PROGRAM prg_Verschalingmetfunctie
VAR
	//POTENTIOMETERRRR
	//0 tot 32767
	nPotentiometer		AT		%I*		:INT;
	nPotentiometerValue		:INT;
	nPower				AT		%Q*		:INT:=32767;
	
	//DISPLAYYYYY
	//–100 tot +2 000
	nDisplay			AT		%Q*		:INT;
END_VAR


//Hier wordt de data van potentiometer van 0 tot 30 verschaald
nPotentiometer:=TO_INT(F_Scale(
	fRawData:= nPotentiometerValue, 
	fRawDataLowerOffLimit:= 0, 
	fRawDataUpperOffLimit:= 32767, 
	fScaleDataLowerOffLimit:= 0, 
	fScaleDataUpperOffLimit:= 10));
	
	
//DUS NU WORDT DE DATA VAN nDisplay van 0 tot 1000 verschaald
nDisplay:=TO_INT(F_Scale(
	fRawData:= nPotentiometer, 
	fRawDataLowerOffLimit:= 0, 
	fRawDataUpperOffLimit:= 10, 
	fScaleDataLowerOffLimit:= 0, 
	fScaleDataUpperOffLimit:= 1000));

END_PROGRAM

(* stored: Version 1.1.0.1, ProductVersion 3.1.4024.15
   POU prg_Verschalingmetfunctie: Id {6c67f3fd-77fc-4cf2-b611-2e0f74a12d4a}, SpecialFunc None *)
